// TIA Portal V20 export
TYPE "typeSequenceControlNodeJobInterface"
// stored: Namespace Unit1.Em6
   STRUCT
      commands { ExternalWritable := 'False'} : "Unit1.Em6.typeSequenceControlNodeJobInterfaceCommands";
      monitoring { ExternalWritable := 'False'} : "Unit1.Em6.typeSequenceControlNodeJobInterfaceMonitoring";
   END_STRUCT;
END_TYPE
